// TIA Portal V19 export
VAR_GLOBAL   // PLC tag table "PROFIsafe Drives"
   Drive_Unit1_TLG30Status AT %I2040.0 : "Safety.LDrvSafe_typeSinaSTlg30Status";   // Safety status word for drive 1   {ExternalWritable false}
   Drive_Unit1_TLG30Control AT %Q2040.0 : "Safety.LDrvSafe_typeSinaSTlg30Control";   // Safety control word for drive 1   {ExternalWritable false}
   Drive_Unit2_TLG30Control AT %Q2047.0 : "Safety.LDrvSafe_typeSinaSTlg30Control";   // Safety control word for drive 2   {ExternalWritable false}
   Drive_Unit2_TLG30Status AT %I2047.0 : "Safety.LDrvSafe_typeSinaSTlg30Status";   // Safety status word for drive 2   {ExternalWritable false}
END_VAR
